PROGRAM Visualaisation_Control
VAR
	mxDebugButton: BOOL;
	mxDebugMode: BOOL;
	mxStationStatus: STRING;
	mxManualMode: BOOL;
END_VAR

IF mxDebugButton THEN
	mxDebugMode:=TRUE;
ELSE
	mxDebugMode:=FALSE;
END_IF

//100:Ready to Work § 200: Getting Booked § 300: Booked and Busy § 400 : Manual mode  § 500: Pause Mode § 1000 : Emergency Mode 
IF gvl.mwStationStatus = 100 THEN
	mxStationStatus:= 'Ready for Order';
	mxManualMode:=FALSE;
ELSIF gvl.mwStationStatus = 200 THEN
	mxStationStatus:= 'Executing booking order from IOStation';
	mxManualMode:=FALSE;
ELSIF gvl.mwStationStatus = 300 THEN
	mxStationStatus:= 'Booked for Order or Busy';
	mxManualMode:=FALSE;
ELSIF gvl.mwStationStatus = 400 THEN
	mxStationStatus:= 'Manual Mode';
	mxManualMode:=TRUE;
ELSIF gvl.mwStationStatus = 500 THEN
	mxStationStatus:= 'Pause Mode';
ELSIF gvl.mwStationStatus = 1000 OR  gvl.ixEmergencyStop THEN
	mxStationStatus:= 'Emergency Mode';
	mxManualMode:=FALSE;
ELSIF gvl.mwStationStatus = 0 THEN
	mxStationStatus:= 'Intial Mode';
	mxManualMode:=FALSE;
ELSIF  gvl.mwStationStatus = 50 THEN
	mxStationStatus:= 'Pre-Condition State';
ELSE
	mxStationStatus:= 'Status Unknown';
END_IF

END_PROGRAM

(* stored: Version 1.1.0.1, ProductVersion 3.1.4024.10
   POU Visualaisation_Control: Id {212f1124-e6e9-482c-9a19-e43dd5520b3d}, SpecialFunc None *)
